FUNCTION_BLOCK FB_CoreVibratoryBowl2
VAR
    iState : INT := 0;
    iState2 : INT := 0;
	FeedbackTimer : TON;
    DelayTimer : TON;
	DelayTimer2 : TON;
END_VAR

CASE iState OF
    0: (* Idle/Off *)
		iState := 10;
	
	10:
        IF GVL_HMI.bSafeties AND GVL_IO.DI_ECS THEN
            iState := iState + 10;
        END_IF

    20: (* Wait for Product in Position *)
		DelayAndAdvance( GVL_InitialSetting.BOWL_RunningDelayTime, iState+1 );
	21:
	    IF GVL_IO.DI_PE3 THEN
            iState := (iState + 10) / 10 * 10;
        END_IF

    30: (* Energize Track Index Solenoid *)
        GVL_IO.DO_PCYL6_E := TRUE;
		DelayAndAdvance( GVL_HMI.i_nPCylinder6ExtendedRunningTime, iState+1 );
	31:
		GVL_IO.DO_PCYL3_E := FALSE;
		iState2 := 0;
		GVL_HMI.i_nCoreCountForStarting := GVL_HMI.i_nCoreCountForStarting + 1;
        iState := (iState + 10) / 10 * 10;
		
	40: (* Check High-Level Sensor *)
		IF GVL_IO.DI_PE6 THEN
			DelayAndAdvance( GVL_HMI.i_nPE6MaintainTime, iState+10 );
		ELSE
			iState := 20;
			DelayTimer.IN := FALSE;
		END_IF
	
	80:
		(* Pause and Wait *)
END_CASE

IF iState >= 20 THEN
	CASE iState2 OF
		0:
			GVL_IO.DO_VB2 := TRUE; 
			IF NOT DelayTimer2.IN THEN
				DelayTimer2(IN := TRUE, PT := INT_TO_TIME(GVL_InitialSetting.VB2_MaintainTime));
			ELSE
				IF DelayTimer2.Q THEN 
					iState2 := iState2 + 10;
				END_IF
			END_IF
		10:
			IF GVL_IO.DI_PE3 THEN
				iState2 := iState2 + 10;
			END_IF
		20:
			(* Stop and Wait *)
	END_CASE
ELSE
	iState2 := 0;
END_IF

METHOD DelayAndAdvance : BOOL
VAR_INPUT
	i_nDelayTime: INT;	// ms
	i_nNextState: INT;
END_VAR

VAR
END_VAR
IF NOT DelayTimer.IN THEN
    DelayTimer(IN := TRUE, PT := INT_TO_TIME(i_nDelayTime));
ELSE
    IF DelayTimer.Q THEN 
        iState := i_nNextState; 
    END_IF
END_IF
END_METHOD

END_FUNCTION_BLOCK

(* stored: Version 1.1.0.1, ProductVersion 3.1.4024.6
   POU FB_CoreVibratoryBowl2: Id {38cac3bb-8f58-4f28-bdcd-b1cc47d57b4f}, SpecialFunc None
   Method DelayAndAdvance: Id {dbec43e2-aff0-447f-9917-a49205f9dcef} *)
